{attribute 'linkalways'} 
{attribute 'no_explicit_call' := 'This FB is a CLASS and must be accessed using methods or properties'}
{attribute 'enable_dynamic_creation'}
FUNCTION_BLOCK _BYTE EXTENDS NumericDatatypeBase
VAR
	localData : BYTE;
	activeData : REFERENCE TO BYTE REF= localData;
END_VAR

PROPERTY PUBLIC Address : PVOID
GET
Address := ADR(activeData);
END_GET
END_PROPERTY

METHOD PUBLIC ClearReference
VAR_INPUT
END_VAR
activeData REF= localData;
END_METHOD

METHOD PUBLIC Clone : I_Datatype
VAR
    pClone : POINTER TO _BYTE;
END_VAR
pClone := __NEW(_BYTE(InitialValue := Value));
Clone := pClone^;
END_METHOD

METHOD FB_init : BOOL
VAR_INPUT
	bInitRetains : BOOL; // if TRUE, the retain variables are initialized (warm start / cold start)
	bInCopyCode : BOOL;  // if TRUE, the instance afterwards gets moved into the copy code (online change)
	InitialValue : BYTE;
END_VAR
localData := InitialValue;
END_METHOD

PROPERTY PUBLIC IsFloat : BOOL
GET
IsFloat := FALSE;
END_GET
END_PROPERTY

PROPERTY PUBLIC IsSigned : BOOL
GET
IsSigned := FALSE;
END_GET
END_PROPERTY

METHOD PUBLIC MakeReferenceTo
VAR_INPUT
	ReferenceTarget : REFERENCE TO BYTE;
END_VAR
activeData REF= ReferenceTarget;
END_METHOD

PROPERTY PUBLIC MaxValue : BYTE
GET
MaxValue := DatatypeLimits.BYTE_MAX_VALUE;
END_GET
END_PROPERTY

PROPERTY PUBLIC MinValue : BYTE
GET
MinValue := DatatypeLimits.BYTE_MIN_VALUE;
END_GET
END_PROPERTY

METHOD PROTECTED SerializeMaxValue
VAR_INPUT
	Serializer : I_Serializer;
END_VAR
Serializer.AddByte(MaxValue);
END_METHOD

METHOD PROTECTED SerializeMinValue
VAR_INPUT
	Serializer : I_Serializer;
END_VAR
Serializer.AddByte(MinValue);
END_METHOD

METHOD PUBLIC SerializeWith
VAR_INPUT
	Serializer : I_Serializer;
END_VAR
Serializer.AddByte(activeData);
END_METHOD

PROPERTY PUBLIC Size : UDINT
GET
Size := SIZEOF(activeData);
END_GET
END_PROPERTY

METHOD TryDeserializeFrom : BOOL
VAR_INPUT
	Deserializer : I_Deserializer;
	Feedback : I_DeserializerFeedback;
END_VAR
TryDeserializeFrom := Deserializer.TryGetByte(activeData, Feedback);
END_METHOD

METHOD TryMakeReferenceTo : BOOL
VAR_INPUT
	Target : I_Datatype;
END_VAR
VAR
	pTargetData : POINTER TO BYTE;
END_VAR
IF NOT (Target.TypeName = TypeName) THEN
	RETURN;
END_IF

pTargetData := Target.Address;
activeData REF= pTargetData^;
TryMakeReferenceTo := TRUE;
END_METHOD

PROPERTY PUBLIC TypeName : T_MAXSTRING
GET
TypeName := 'BYTE';
END_GET
END_PROPERTY

PROPERTY PUBLIC Value : REFERENCE TO BYTE
GET
Value REF= activeData;
END_GET
END_PROPERTY

END_FUNCTION_BLOCK

(* stored: Version 1.1.0.1, ProductVersion 3.1.4024.12
   POU _BYTE: Id {015fee84-30df-4efb-96c8-fa65eaa5aa83}, SpecialFunc None
   Folder Constructor: Id {52a26577-a6bc-4aa5-9ef8-f187627d1642}
   Folder Protected: Id {8aa9057a-15bb-4079-bf78-cfd21590127a}
   Property Address: Id {f4658331-4fdd-43d9-be9e-00542c59946a}
   Get Get: Id {d753ed97-43be-40c2-a48d-d6d299103d65}
   Method ClearReference: Id {3854d391-b7b2-4b47-9f9a-18e69b0dcbda}
   Method Clone: Id {e218fd2c-90c0-45b2-a3dc-c3ce9829dc9a}
   Method FB_init: Id {c73f40e7-da83-43bf-b9c3-680c5d3df281}
   Property IsFloat: Id {65b20559-d076-483f-b3d3-9f65fcb52652}
   Get Get: Id {e8ca72cd-2c65-4183-94e9-64387bc9c4f2}
   Property IsSigned: Id {83a3b0ce-180f-4907-989b-f922d0f2214e}
   Get Get: Id {d6690cbf-d958-4d50-9841-8375714a31ff}
   Method MakeReferenceTo: Id {18ec47ae-83dd-4afc-a3f0-890a89595ae0}
   Property MaxValue: Id {47ded2cf-bef0-4212-afe1-d53ae7a8073a}
   Get Get: Id {be9751fc-c4c7-4b02-b040-d761b9f03f84}
   Property MinValue: Id {b0a5acb4-937e-49e0-ae6b-7185073a6fe6}
   Get Get: Id {8b359cfc-8c76-478a-a1b9-a2dfcc7188e4}
   Method SerializeMaxValue: Id {2b2dd19b-d33d-47a5-a3fd-8f7871724ec3}
   Method SerializeMinValue: Id {6bd0c9eb-7393-4705-994d-fa6038d95d76}
   Method SerializeWith: Id {66fb1589-93aa-48cc-9b7f-87181c23e74d}
   Property Size: Id {7f95387a-676f-4254-8a17-a3b6e9673cda}
   Get Get: Id {128d205a-ce0d-44fe-9ee1-7b8137c3ed50}
   Method TryDeserializeFrom: Id {ed654a62-7512-4173-bcd9-55f451d1c2af}
   Method TryMakeReferenceTo: Id {dc7c26da-384c-431a-824b-f41d2d332124}
   Property TypeName: Id {1c1c2320-0402-4c90-bee9-948e0946fa55}
   Get Get: Id {2f3ac17e-d722-4c9a-a69e-7923adb5d499}
   Property Value: Id {2e144ab6-c08f-45e7-82aa-2cda5774589e}
   Get Get: Id {43823d97-4013-4032-a00f-d395ded07007} *)
